TYPE ST_SafetyStatus :
STRUCT
END_STRUCT
END_TYPE

(* stored: Version 1.1.0.1, ProductVersion 3.1.4024.11
   DUT ST_SafetyStatus: Id {e9853b14-b0c3-4bf2-92c4-c725f4c85a2f} *)
